{attribute 'linkalways'} 
{attribute 'no_explicit_call' := 'This FB is a CLASS and must be accessed using methods or properties'}
{attribute 'enable_dynamic_creation'}
FUNCTION_BLOCK FINAL MIN_DINT EXTENDS Node
VAR
	in1 : _DINT(0);
	in2 : _DINT(0);
	out : _DINT(0);
END_VAR

METHOD PUBLIC Clone : I_Node
VAR
	pNode : POINTER TO MIN_DINT;
END_VAR
pNode := __NEW(MIN_DINT);
Clone := pNode^;
END_METHOD

METHOD FB_init : BOOL
VAR_INPUT
	bInitRetains : BOOL; // if TRUE, the retain variables are initialized (warm start / cold start)
	bInCopyCode : BOOL;  // if TRUE, the instance afterwards gets moved into the copy code (online change)
END_VAR
AddInput('in1',THIS^.in1);
AddInput('in2',THIS^.in2);
AddOutput('out', THIS^.out);
END_METHOD

METHOD PROTECTED OnExecute
VAR
END_VAR
out.Value := MIN(in1.Value, in2.Value);
END_METHOD

END_FUNCTION_BLOCK

(* stored: Version 1.1.0.1, ProductVersion 3.1.4024.15
   POU MIN_DINT: Id {59073f62-dfce-4907-9a71-fabb8bbcf863}, SpecialFunc None
   Folder Constructor: Id {a1437632-a603-44f5-b12f-14dd13471654}
   Method Clone: Id {a96959fe-d3e6-4213-94b5-22fe9531ece3}
   Method FB_init: Id {b03a2a0a-eb16-4835-9307-0ead8fe9b790}
   Method OnExecute: Id {df8ad0ae-5898-41d9-9088-bb86ebc74649} *)
